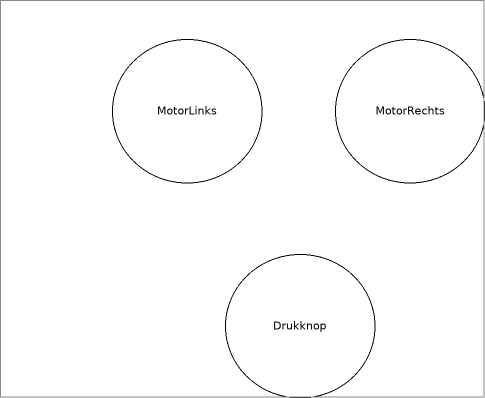
VISUALIZATION Visualization_MotorMetDrukknop  // 485x398
    Ellipse (112,39 150x144), "MotorLinks", colour toggle: prg_MotorMetDrukknop.MotorLinks
    Ellipse (225,254 150x144), "Drukknop"
        tap prg_MotorMetDrukknop.Drukknop
    Ellipse (335,39 150x144), "MotorRechts", colour toggle: prg_MotorMetDrukknop.MotorRechts
END_VISUALIZATION

(* stored: Version 1.1.0.1, ProductVersion 3.1.4024.15
   Visu Visualization_MotorMetDrukknop: Id {af7e264f-0b3c-43c2-819a-4e61a00c5b75} *)
